# EPICS substitutions: db/user.substitutions
# Example substitutions file

file "db/dbExample1.db" {
    { user = "lees" }
}

file db/dbExample2.db {
    pattern { user, no, scan }
        { "lees", 1, "1 second" }
        { "lees", 2, "2 second" }
        { "lees", 3, "5 second" }
}
